FUNCTION_BLOCK Controller
  (* Standard: 61499-2 *)
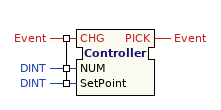
  EVENT_INPUT
    CHG WITH NUM, SetPoint;
  END_EVENT
  EVENT_OUTPUT
    PICK;
  END_EVENT
  VAR_INPUT
    NUM : DINT;
    SetPoint : DINT;
  END_VAR
  VAR
    match : BOOL;
  END_VAR
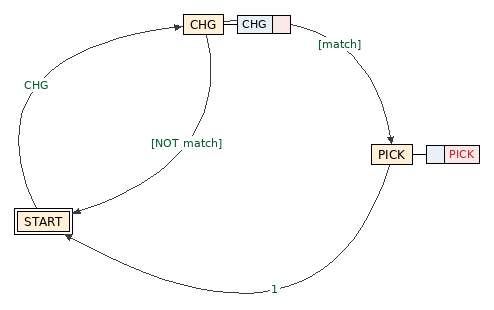
  EC_STATES
    START;
    CHG : CHG;
    PICK : -> PICK;
  END_STATES
  EC_TRANSITIONS
    START TO CHG := CHG;
    CHG TO START := [NOT match];
    PICK TO START := 1;
    CHG TO PICK := [match];
  END_TRANSITIONS
  ALGORITHM CHG IN ST:
match := (NUM = SetPoint);&#10;
  END_ALGORITHM
END_FUNCTION_BLOCK
